FUNCTION_BLOCK  Vision_StateMachine
VAR
//var to get struct data from ck_real_value function
cx_vision_data : ck_real_flag_data;
cy_vision_data : ck_real_flag_data;
nut_turn_data : ck_real_flag_data;

sep_pos_data : ck_real_flag_data;

sep_rot_rigth_data :ck_real_flag_data;
sep_rot_left_data :ck_real_flag_data;


//internal aux state
I_STATE : INT:=-1;
END_VAR

VAR_INPUT
init_: BOOL:= FALSE;
//global aux state
G_STATE: INT:=-1;

END_VAR


VAR_OUTPUT
	State_complete : BOOL:= FALSE;
	Act_Gl_State :INT:=-1;
	Act_In_State: INT:=-1;
END_VAR

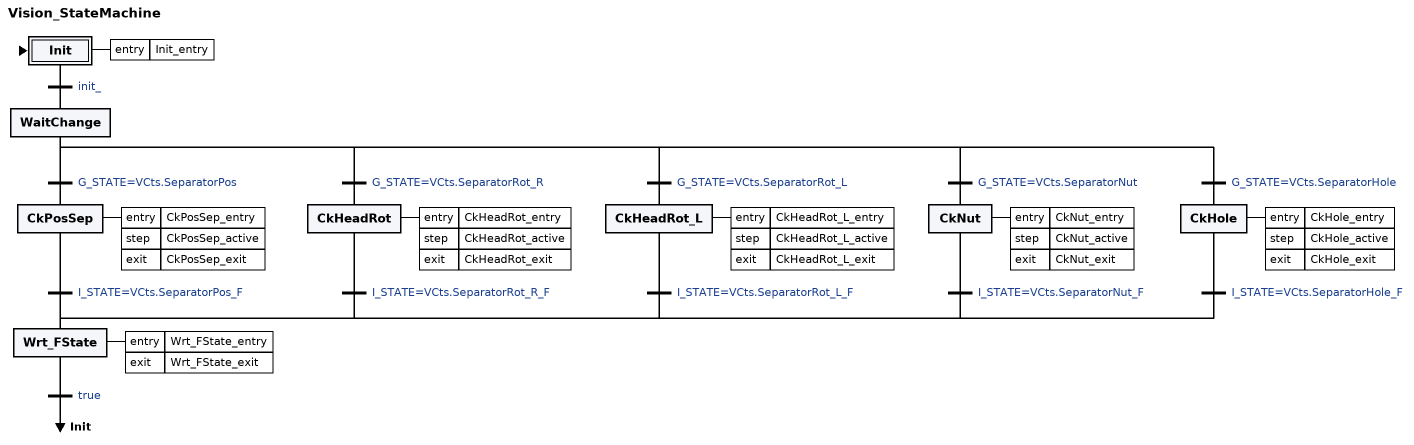
INITIAL_STEP Init:
    Init_entry(P1);  // entry action
END_STEP
TRANSITION FROM Init TO WaitChange
    := init_;
END_TRANSITION
STEP WaitChange:
END_STEP
TRANSITION FROM WaitChange TO CkPosSep
    := G_STATE=VCts.SeparatorPos;
END_TRANSITION
STEP CkPosSep:
    CkPosSep_entry(P1);  // entry action
    CkPosSep_active(N);  // step action
    CkPosSep_exit(P0);  // exit action
END_STEP
TRANSITION FROM CkPosSep TO Wrt_FState
    := I_STATE=VCts.SeparatorPos_F;
END_TRANSITION
TRANSITION FROM WaitChange TO CkHeadRot
    := G_STATE=VCts.SeparatorRot_R;
END_TRANSITION
STEP CkHeadRot:
    CkHeadRot_entry(P1);  // entry action
    CkHeadRot_active(N);  // step action
    CkHeadRot_exit(P0);  // exit action
END_STEP
TRANSITION FROM CkHeadRot TO Wrt_FState
    := I_STATE=VCts.SeparatorRot_R_F;
END_TRANSITION
TRANSITION FROM WaitChange TO CkHeadRot_L
    := G_STATE=VCts.SeparatorRot_L;
END_TRANSITION
STEP CkHeadRot_L:
    CkHeadRot_L_entry(P1);  // entry action
    CkHeadRot_L_active(N);  // step action
    CkHeadRot_L_exit(P0);  // exit action
END_STEP
TRANSITION FROM CkHeadRot_L TO Wrt_FState
    := I_STATE=VCts.SeparatorRot_L_F;
END_TRANSITION
TRANSITION FROM WaitChange TO CkNut
    := G_STATE=VCts.SeparatorNut;
END_TRANSITION
STEP CkNut:
    CkNut_entry(P1);  // entry action
    CkNut_active(N);  // step action
    CkNut_exit(P0);  // exit action
END_STEP
TRANSITION FROM CkNut TO Wrt_FState
    := I_STATE=VCts.SeparatorNut_F;
END_TRANSITION
TRANSITION FROM WaitChange TO CkHole
    := G_STATE=VCts.SeparatorHole;
END_TRANSITION
STEP CkHole:
    CkHole_entry(P1);  // entry action
    CkHole_active(N);  // step action
    CkHole_exit(P0);  // exit action
END_STEP
TRANSITION FROM CkHole TO Wrt_FState
    := I_STATE=VCts.SeparatorHole_F;
END_TRANSITION
STEP Wrt_FState:
    Wrt_FState_entry(P1);  // entry action
    Wrt_FState_exit(P0);  // exit action
END_STEP
TRANSITION FROM Wrt_FState TO Init
    := true;
END_TRANSITION

ACTION CkHeadRot_active:

//read register from robot and chek is can read 2 or more correct values 
IF ck_state_v(VCts.SeparatorRot_R_I) THEN
	 I_STATE:= VCts.SeparatorRot_R_I;

//verifies that the vision system has completed its task
ELSIF ck_state_v(VCts.SeparatorRot_R_F) THEN
	//read the values processed by the vision system and send to robot
	sep_rot_rigth_data := ck_real_value(Vision_struct.Head_rigth_value);
	//check if all values are correct
	IF sep_rot_rigth_data.Flag THEN
		//write variables from PLC to CS.UR5 Robot
		IF wr_real_value(VCts.HEAD_RIGTH_VALUE,sep_rot_rigth_data.Value) THEN
			I_STATE := VCts.SeparatorRot_R_F;

		END_IF
	END_IF
	
END_IF


//read internal variable and write over output variable
Act_In_State := I_STATE;
END_ACTION

ACTION CkHeadRot_entry:

//start the vision system
wr_state_v(Vcts.SeparatorRot_R);

//write the retain state variable 
Act_Gl_State:=VCts.SeparatorRot_R;
END_ACTION

ACTION CkHeadRot_exit:
//write reset state variables to visiom system.
wr_state_v(RCts.RESET_STATE);
//reset Global state variable
G_STATE := -1;
I_STATE :=-1;
END_ACTION

ACTION CkHeadRot_L_active:

//read register from robot and chek is can read 2 or more correct values 
IF ck_state_v(VCts.SeparatorRot_L_I) THEN
	 I_STATE:= VCts.SeparatorRot_L_I;
//verifies that the vision system has completed its task
ELSIF ck_state_v(VCts.SeparatorRot_L_F) THEN
	//read the values processed by the vision system and send to robot
	sep_rot_left_data := ck_real_value(Vision_struct.Head_left_value);
	//check if all values are correct
	IF sep_rot_left_data.Flag THEN
		//write variables from PLC to CS.UR5 Robot
		IF wr_real_value(VCts.HEAD_LEFT_VALUE,sep_rot_left_data.Value) THEN
			I_STATE := VCts.SeparatorRot_L_F;
		END_IF
	END_IF
	
END_IF


//read internal variable and write over output variable
Act_In_State := I_STATE;
END_ACTION

ACTION CkHeadRot_L_entry:
//start the vision system
wr_state_v(Vcts.SeparatorRot_L);

//write the retain state variable 
Act_Gl_State:=VCts.SeparatorRot_L;
END_ACTION

ACTION CkHeadRot_L_exit:
//write reset state variables to visiom system.
wr_state_v(RCts.RESET_STATE);
//reset Global state variable
G_STATE := -1;
END_ACTION

ACTION CkHole_active:
//read register from robot and chek is can read 2 or more correct values 
IF ck_state_v(VCts.SeparatorHole_I) THEN
	 I_STATE:= VCts.SeparatorHole_I;
//verifies that the vision system has completed its task
ELSIF ck_state_v(VCts.SeparatorHole_F) THEN
	//read the values processed by the vision system and send to robot
	cx_vision_data := ck_real_value(Vision_struct.Cx_value_hole);
	cy_vision_data := ck_real_value(Vision_struct.Cy_value_hole);
	//check if all values are correct
	IF cx_vision_data.Flag AND cy_vision_data.Flag THEN
		//write variables from PLC to CS.UR5 Robot
		IF wr_real_value(VCts.CX_VALUE,cx_vision_data.Value) THEN
			IF wr_real_value(VCts.CY_VALUE,cy_vision_data.Value) THEN				
						I_STATE := VCts.SeparatorNut_F;
			END_IF
		
		END_IF
	END_IF
	
END_IF




//read internal variable and write over output variable
Act_In_State := I_STATE;
END_ACTION

ACTION CkHole_entry:
//start the vision system
wr_state_v(Vcts.SeparatorNut);

//write the retain state variable 
Act_Gl_State:=VCts.SeparatorNut;
END_ACTION

ACTION CkHole_exit:
//write reset state variables to visiom system.
wr_state_v(RCts.RESET_STATE);
//reset Global state variable
G_STATE := -1;
END_ACTION

ACTION CkNut_active:


//read register from robot and chek is can read 2 or more correct values 
IF ck_state_v(VCts.SeparatorNut_I) THEN
	 I_STATE:= VCts.SeparatorNut_I;
//verifies that the vision system has completed its task
ELSIF ck_state_v(VCts.SeparatorNut_F) THEN
	//read the values processed by the vision system and send to robot
	cx_vision_data := ck_real_value(Vision_struct.Cx_value_nut);
	cy_vision_data := ck_real_value(Vision_struct.Cy_value_nut);
	nut_turn_data := ck_real_value(Vision_struct.Nut_turn_value);
	//check if all values are correct
	IF cx_vision_data.Flag AND cy_vision_data.Flag AND nut_turn_data.Flag THEN
		//write variables from PLC to CS.UR5 Robot
		IF wr_real_value(VCts.CX_VALUE,cx_vision_data.Value) THEN
			IF wr_real_value(VCts.CY_VALUE,cy_vision_data.Value) THEN
				IF wr_real_value(VCts.NUT_VALUE,nut_turn_data.Value) THEN
						I_STATE := VCts.SeparatorNut_F;
				END_IF
			END_IF
		
		END_IF
	END_IF
	
END_IF



//read internal variable and write over output variable
Act_In_State := I_STATE;
END_ACTION

ACTION CkNut_entry:
//start the vision system
wr_state_v(Vcts.SeparatorNut);

//write the retain state variable 
Act_Gl_State:=VCts.SeparatorNut;
END_ACTION

ACTION CkNut_exit:
//write reset state variables to visiom system.
wr_state_v(RCts.RESET_STATE);
//reset Global state variable
G_STATE := -1;
END_ACTION

ACTION CkPosSep_active:

//read register from robot and chek is can read 2 or more correct values 
IF ck_state_v(VCts.SeparatorPos_I) THEN
	 I_STATE:= VCts.SeparatorPos_I;
	
//verifies that the vision system has completed its task
ELSIF ck_state_v(VCts.SeparatorPos_F) THEN
	//read the values processed by the vision system and send to robot
	sep_pos_data := ck_real_value(Vision_struct.Pos_sep);
	//check if all values are correct
	IF sep_pos_data.Flag THEN
		//write variables from PLC to CS.UR5 Robot
		IF wr_real_value(VCts.SEP_POS_VALUE,sep_pos_data.Value) THEN
			I_STATE := VCts.SeparatorPos_F;
	
		END_IF
	END_IF
	
END_IF

//read internal variable and write over output variable
Act_In_State := I_STATE;
END_ACTION

ACTION CkPosSep_entry:

//start the vision system
wr_state_v(Vcts.SeparatorPos);

//write the retain state variable 
Act_Gl_State:=VCts.SeparatorPos;
END_ACTION

ACTION CkPosSep_exit:

//write reset state variables to visiom system.
wr_state_v(RCts.RESET_STATE);
//reset Global state variable
G_STATE := -1;
//rest internat state variable
I_STATE :=-1;
END_ACTION

ACTION Init_entry:
//write output variable to indicate that the robot execute the state 
State_complete := FALSE;
init_:=FALSE;
G_STATE := -1;
I_STATE :=-1;
END_ACTION

ACTION Wrt_FState_entry:
//write output variable to indicate that the robot execute the state 
State_complete := TRUE;
END_ACTION

ACTION Wrt_FState_exit:
//write output variable to indicate that the robot execute the state 
State_complete := FALSE;
init_:=FALSE;

G_STATE := -1;
//rest internat state variable
I_STATE :=-1;
END_ACTION

END_FUNCTION_BLOCK

(* stored: Version 1.1.0.1, ProductVersion 3.1.4024.4
   POU Vision_StateMachine: Id {f93bb11a-f5cd-40ad-a452-b50656e25a24}, SpecialFunc None
   Action CkHeadRot_active: Id {79483949-fdb1-43c7-85b0-66a3b8676161}
   Action CkHeadRot_entry: Id {7ebbfc85-5aad-4741-9c48-8a8ecd05823e}
   Action CkHeadRot_exit: Id {8e1964bb-4c65-4438-8d8b-94b34bd867af}
   Action CkHeadRot_L_active: Id {711619a1-95dc-453c-8399-d35c9e24aa1f}
   Action CkHeadRot_L_entry: Id {e7280780-b5cc-4cfa-a7ac-92dc66778b28}
   Action CkHeadRot_L_exit: Id {65a68dea-7154-4042-86c2-12ba9be18eca}
   Action CkHole_active: Id {1c91934e-b1c9-4f07-a4c3-8849aee832cd}
   Action CkHole_entry: Id {ee9a1cea-e91f-4e21-b1ae-6ae94fbf405e}
   Action CkHole_exit: Id {15f08814-3d85-42b8-8bef-93215c40194e}
   Action CkNut_active: Id {a76c4aea-c03d-4f2e-a27c-e3588e7a8d51}
   Action CkNut_entry: Id {7b639d02-350f-49a2-9682-bc001a1885d5}
   Action CkNut_exit: Id {d8ded961-8fc2-4dab-9fb9-edf8d208d7d5}
   Action CkPosSep_active: Id {5eb9aaf2-ba77-4c72-8011-fd3d40ba003d}
   Action CkPosSep_entry: Id {90dd64f5-3a3d-4fd1-ac87-8dfd3a83d6a7}
   Action CkPosSep_exit: Id {b8d496af-bbe4-4811-b6ee-ef9fbec01c2f}
   Action Init_entry: Id {3914e7b7-2735-4d32-afc2-e796baedcd53}
   Action Wrt_FState_entry: Id {1d35addc-fc6f-4851-a277-1b750685bb69}
   Action Wrt_FState_exit: Id {0894eb1e-4132-45ea-bf48-d140c510b14e} *)
